METHOD PROTECTED OnStart
IF __ISVALIDREF(inoStatus) THEN
    THIS^.inoStatus.ActionDescription := '<#Separator task started.#>';
END_IF;

_componentReady := false;
CallTimers(FALSE);
END_METHOD

(*~
    <docu>
        <summary>
            Restores this instance to the Ready state. Can be called explicitly or from within one of the restore mechanisms.
            <para>
                See also <see cref="PlcDocu.TcoCore.TcoTask.AutoRestorable()"/>
            </para>
        </summary>
    </docu>
~*)
METHOD Restore : ITcoRestorable
SUPER^.Restore();
_componentReady := false;
END_METHOD

END_FUNCTION_BLOCK

// ---- POUs/Prototypes/TixonVibro/TcoTixonVibro_v_1_x_x.TcPOU
FUNCTION_BLOCK TcoTixonVibro_v_1_x_x EXTENDS TcoCore.TcoComponent
VAR_INPUT
    inControllerInAuto : BOOL;
    inNotEmptyFeeder : BOOL;
    inSeparatorHomePos : BOOL;
    inFillingSensor : BOOL;
    inSeparatorPresent : BOOL;
    inComponentOutOfBox : BOOL;
    inSeparatorWorkPos : BOOL;
END_VAR
VAR_OUTPUT
    outFeedingA : BOOL;
    outSepareComponent : BOOL;
    outBlowValveA : BOOL;
    outRedLed : BOOL;
    outGreenLed : BOOL;
    outHopper : BOOL;
    outShotComponent : BOOL;
END_VAR
VAR
    {attribute addProperty Name "<#Status#>"}
    {attribute clr [ReadOnly()]}
    _status : TcoTixonVibro_Status_v_1_x_x;
    {attribute addProperty Name "<#Control#>"}
    _control : TcoTixonVibro_Control_v_1_x_x;
    {attribute addProperty Name "<#Config#>"}
    _config : TcoTixonVibro_Config_v_1_x_x;
    _someTaskIsActive : BOOL;
    {attribute 'hide'}
    _blink : TcoUtilities.TcoBlinker(THIS^);
    _runAutomatic : BOOL;
    _hasError : BOOL;
END_VAR
VAR
    {attribute addProperty Name "<#Separator task#>"}
    _separatorTask : TcoTixonVibroSeparatorTask(THIS^);
    {attribute addProperty Name "<#Buffer task#>"}
    _bufferTask : TcoTixonBufferTask(THIS^);
    {attribute addProperty Name "<#Hopper task#>"}
    _hopperTask : TcoTixonHopperTask(THIS^);
    {attribute addProperty Name "<#Restore#>"}
    _restoreTask : TcoCore.TcoTask(THIS^);
END_VAR
VAR
    {attribute 'hide'}
    _sb : TcoCore.StringBuilder;
END_VAR

_blink(inOnTime := _config.BlinkTime, inOffTime := _config.BlinkTime);
UpdateStatus();
_separatorTask.Enabled := TRUE;
_separatorTask.ErrorTime := _config.ErrorTimeSeparator;
_separatorTask(inoConfig := _config, inoControl := _control, inoStatus := _status);
_bufferTask.Enabled := TRUE;
_bufferTask.ErrorTime := _config.ErrorTimeBuffer;
_bufferTask(inoConfig := _config, inoControl := _control, inoStatus := _status);
_hopperTask.ErrorTime := _config.ErrorTimeHopper;
_hopperTask.Enabled := _config.HopperActive;
_hopperTask(inoConfig := _config, inoControl := _control, inoStatus := _status);
//*************RESTORE********************
_restoreTask.Enabled := TRUE;

IF _restoreTask.Execute() THEN
    Restore();
    _restoreTask.DoneWhen(TRUE);
END_IF
//****************************************
UpdateControl();

METHOD PUBLIC BufferFeed : TcoCore.ITcoTaskStatus
BufferFeed := _bufferTask.Invoke();
_bufferTask.AutoRestore := false;
END_METHOD

PROPERTY PUBLIC BufferTask : REFERENCE TO TcoTixonBufferTask
GET
BufferTask ref= _bufferTask;
END_GET
END_PROPERTY

(*~
    <docu>
        <summary>
            Gets the configuration of the Tixon Vibro.
        </summary>
    </docu>
~*)
PROPERTY Config : REFERENCE TO TcoTixonVibro_Config_v_1_x_x
GET
Config REF= _config;
END_GET
END_PROPERTY

METHOD PUBLIC CyclicBufferFeed : TcoCore.ITcoTaskStatus
CyclicBufferFeed := _bufferTask.Invoke();
_bufferTask.AutoRestore := true;
END_METHOD

METHOD PUBLIC CyclicHopperFeed : TcoCore.ITcoTaskStatus
CyclicHopperFeed := _hopperTask.Invoke();
_hopperTask.AutoRestore := TRUE;
END_METHOD

METHOD PUBLIC CyclicSepare : TcoCore.ITcoTaskStatus
CyclicSepare := _separatorTask.Invoke();
_separatorTask.AutoRestore := true;
END_METHOD

METHOD PUBLIC DefaultSignalisation
VAR_INPUT
END_VAR
// led signalisation
_hasError := _separatorTask.Error OR _bufferTask.Error OR _hopperTask.Error;
_control.GreenLed := FALSE;
_control.RedLed := FALSE;

IF NOT _status.ControllerInAuto THEN
    _control.GreenLed := TRUE;
    _control.RedLed := TRUE;
ELSIF _hasError AND _blink.IsOn AND _status.ControllerInAuto THEN
    _control.RedLed := TRUE;
ELSIF _status.ControllerInAuto AND NOT _hasError AND _status.NotEmptyFeeder THEN
    _control.GreenLed := TRUE;
ELSIF _blink.IsOn AND _status.ControllerInAuto AND NOT _status.NotEmptyFeeder THEN
    _control.GreenLed := TRUE;
    _control.RedLed := TRUE;
END_IF
END_METHOD

METHOD PUBLIC HopperFeed : TcoCore.ITcoTaskStatus
HopperFeed := _hopperTask.Invoke();
_hopperTask.AutoRestore := false;
END_METHOD

PROPERTY PUBLIC HopperTask : reference TO TcoTixonHopperTask
GET
HopperTask ref= _hopperTask;
END_GET
END_PROPERTY

METHOD PUBLIC Push
VAR_INPUT
    inReqOn : BOOL;
END_VAR
_control.ShotComponent := inReqOn;
END_METHOD

(*~
    <docu>
        <summary>
            Restores this instance to the Ready state. Can be called explicitly or from within one of the restore mechanisms.
        </summary>
    </docu>
~*)
METHOD Restore : ITcoRestorable
RestoreTasks();
_control.BlowAValve := FALSE;
_control.FeedingA := FALSE;
_control.GreenLed := FALSE;
_control.RedLed := FALSE;
_control.SepareComponent := FALSE;
_control.ShotComponent := FALSE;
_control.Hooper := FALSE;
END_METHOD

METHOD INTERNAL RestoreTasks
_separatorTask.Restore();
_bufferTask.Restore();
_hopperTask.Restore();
END_METHOD

PROPERTY PUBLIC SeparatorTask : REFERENCE TO TcoTixonVibroSeparatorTask
GET
SeparatorTask ref= _separatorTask;
END_GET
END_PROPERTY

METHOD PUBLIC Separe : TcoCore.ITcoTaskStatus
Separe := _separatorTask.Invoke();
_separatorTask.AutoRestore := false;
END_METHOD

(*~
    <docu>
        <summary>
            Custom service (manual, maintenance) logic.
            This method must be implemented in derived class.
        </summary>
    </docu>
~*)
METHOD PROTECTED ServiceMode
END_METHOD

(*~
    <docu>
        <summary>
            Gets the status of the Tixon Vibro.
        </summary>
    </docu>
~*)
PROPERTY Status : REFERENCE TO TcoTixonVibro_Status_v_1_x_x
GET
Status REF= _status;
END_GET
END_PROPERTY

METHOD INTERNAL UpdateControl
VAR_INPUT
END_VAR
VAR
    index : INT;
END_VAR
outBlowValveA := _control.BlowAValve;
outFeedingA := _control.FeedingA;
outGreenLed := _control.GreenLed;
outRedLed := _control.RedLed;
outSepareComponent := _control.SepareComponent;
outShotComponent := _control.ShotComponent;
outHopper := _control.Hooper;
END_METHOD

METHOD INTERNAL UpdateStatus
VAR
END_VAR
_status.ComponentOutOfBox := inComponentOutOfBox;
_status.NotEmptyFeeder := inNotEmptyFeeder;
_status.FillingSensor := inFillingSensor;
_status.SeparatorHomePos := inSeparatorHomePos;
_status.SeparatorPresent := inSeparatorPresent;
_status.ControllerInAuto := inControllerInAuto;
_status.SeparatorWorkPos := inSeparatorWorkPos;
END_METHOD

END_FUNCTION_BLOCK
